FUNCTION_BLOCK FB_Plant
VAR_INPUT
	fControlInput		: REAL;
END_VAR
VAR_OUTPUT
	fActualOutput		: REAL;
END_VAR
VAR
	fbPart1				: FB_PT1 := (fT1 := T#3S);
	fbPart2				: FB_PT1 := (fP := 2.4, fT1 := T#10s);				
END_VAR


fbPart1(
	fInput := fControlInput
);

fbPart2(
	fInput := fbPart1.fOutput
);

fActualOutput := fbPart2.fOutput;

END_FUNCTION_BLOCK

(* stored: Version 1.1.0.1, ProductVersion 3.1.4022.10
   POU FB_Plant: Id {707443b2-b8a8-492f-9046-0ace2b83d533}, SpecialFunc None *)
